# EPICS substitutions: ek9000App/Db/EL1012.substitutions
file EL1012.template
{ 	pattern
	{
		TERMINAL,

	}
	{
	}
}
